FUNCTION_BLOCK fb_gm_operationElecylinder
VAR_INPUT
END_VAR
VAR_OUTPUT
END_VAR
VAR
	SFCInit: bool;
	TranPosDone: BOOL;
	TranNegDone: BOOL;
	flgInitDone: BOOL;
	PickUpPosDone: BOOL;
	PickUpNegDone: BOOL;
	var_process: INT;
END_VAR

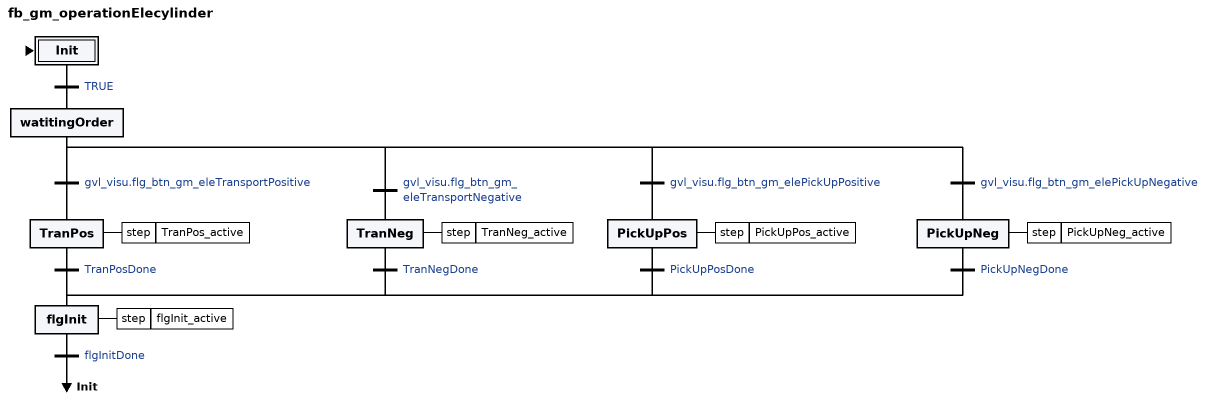
INITIAL_STEP Init:
END_STEP
TRANSITION FROM Init TO watitingOrder
    := TRUE;
END_TRANSITION
STEP watitingOrder:
END_STEP
TRANSITION FROM watitingOrder TO TranPos
    := gvl_visu.flg_btn_gm_eleTransportPositive;
END_TRANSITION
STEP TranPos:
    TranPos_active(N);  // step action
END_STEP
TRANSITION FROM TranPos TO flgInit
    := TranPosDone;
END_TRANSITION
TRANSITION FROM watitingOrder TO TranNeg
    := gvl_visu.flg_btn_gm_eleTransportNegative;
END_TRANSITION
STEP TranNeg:
    TranNeg_active(N);  // step action
END_STEP
TRANSITION FROM TranNeg TO flgInit
    := TranNegDone;
END_TRANSITION
TRANSITION FROM watitingOrder TO PickUpPos
    := gvl_visu.flg_btn_gm_elePickUpPositive;
END_TRANSITION
STEP PickUpPos:
    PickUpPos_active(N);  // step action
END_STEP
TRANSITION FROM PickUpPos TO flgInit
    := PickUpPosDone;
END_TRANSITION
TRANSITION FROM watitingOrder TO PickUpNeg
    := gvl_visu.flg_btn_gm_elePickUpNegative;
END_TRANSITION
STEP PickUpNeg:
    PickUpNeg_active(N);  // step action
END_STEP
TRANSITION FROM PickUpNeg TO flgInit
    := PickUpNegDone;
END_TRANSITION
STEP flgInit:
    flgInit_active(N);  // step action
END_STEP
TRANSITION FROM flgInit TO Init
    := flgInitDone;
END_TRANSITION

ACTION flgInit_active:
IF flgInit._x AND flgInit.x = FALSE THEN
	flgInitDone:= FALSE;
	gvl_visu.flg_btn_gm_eleTransportPositive := FALSE;
	gvl_visu.flg_btn_gm_eleTransportNegative := FALSE;
	gvl_visu.flg_btn_gm_elePickUpPositive := FALSE;
	gvl_visu.flg_btn_gm_elePickUpNegative := FALSE;
	gvl_visu.flg_btn_eleSamplePositive := FALSE;
	gvl_visu.flg_btn_eleSampleNegative := FALSE;
	gvl_visu.flg_btn_eleTrayChangePositive := FALSE;
	gvl_visu.flg_btn_eleTrayChangeNegative := FALSE;
	gvl_visu.flg_btn_eleRotaryPositive := FALSE;
	gvl_visu.flg_btn_eleRotaryNegative := FALSE;
ELSIF flgInit._x AND flgInit.x THEN
	flgInitDone := TRUE;
END_IF
END_ACTION

PROPERTY p_Init : bool
GET
p_init := THIS^.SFCInit;
END_GET
SET
THIS^.SFCInit := p_init;
END_SET
END_PROPERTY

ACTION PickUpNeg_active:
IF PickUpNeg._x AND PickUpNeg.x = FALSE THEN
	PickUpNegDone := FALSE;
	gvl_elecylinder.fbi_gm_axisPickUp.in_flg_run := FALSE;
	gvl_elecylinder.fbi_gm_axisPickUp.in_var_moveMode := eP_eleMoveMode.eleA;
	var_process := 0;
ELSIF PickUpNeg._x AND PickUpNeg.x THEN
	CASE var_process OF
		0:
			gvl_elecylinder.fbi_gm_axisPickUp.in_flg_run := TRUE;
			var_process := 1;
		1:
			IF gvl_elecylinder.fbi_gm_axisPickUp.out_flg_Done THEN
				gvl_elecylinder.fbi_gm_axisPickUp.in_flg_run := FALSE;
				PickUpNegDone := TRUE;
			END_IF
	END_CASE
END_IF
END_ACTION

ACTION PickUpPos_active:
IF PickUpPos._x AND PickUpPos.x = FALSE THEN
	PickUpPosDone := FALSE;
	gvl_elecylinder.fbi_gm_axisPickUp.in_flg_run := FALSE;
	gvl_elecylinder.fbi_gm_axisPickUp.in_var_moveMode := eP_eleMoveMode.eleB;
	var_process := 0;
ELSIF PickUpPos._x AND PickUpPos.x THEN
	CASE var_process OF
		0:
			gvl_elecylinder.fbi_gm_axisPickUp.in_flg_run := TRUE;
			var_process := 1;
		1:
			IF gvl_elecylinder.fbi_gm_axisPickUp.out_flg_Done THEN
				gvl_elecylinder.fbi_gm_axisPickUp.in_flg_run := FALSE;
				PickUpPosDone := TRUE;
			END_IF
	END_CASE
END_IF
END_ACTION

ACTION TranNeg_active:
IF TranNeg._x AND TranNeg.x = FALSE THEN
	TranNegDone := FALSE;
	gvl_elecylinder.fbi_gm_axisTransport.in_flg_run := FALSE;
	gvl_elecylinder.fbi_gm_axisTransport.in_var_moveMode := eP_eleMoveMode.eleA;
	var_process := 0;
ELSIF TranNeg._x AND TranNeg.x THEN
	CASE var_process OF
		0:
			gvl_elecylinder.fbi_gm_axisTransport.in_flg_run := TRUE;
			var_process := 1;
		1:
			IF gvl_elecylinder.fbi_gm_axisTransport.out_flg_Done THEN
				gvl_elecylinder.fbi_gm_axisTransport.in_flg_run := FALSE;
				TranNegDone := TRUE;
			END_IF
	END_CASE
END_IF
END_ACTION

ACTION TranPos_active:
IF TranPos._x AND TranPos.x = FALSE THEN
	TranPosDone := FALSE;
	gvl_elecylinder.fbi_gm_axisTransport.in_flg_run := FALSE;
	gvl_elecylinder.fbi_gm_axisTransport.in_var_moveMode := eP_eleMoveMode.eleB;
	var_process := 0;
ELSIF TranPos._x AND TranPos.x THEN
	CASE var_process OF
		0:
			gvl_elecylinder.fbi_gm_axisTransport.in_flg_run := TRUE;
			var_process := 1;
		1:
			IF gvl_elecylinder.fbi_gm_axisTransport.out_flg_Done THEN
				gvl_elecylinder.fbi_gm_axisTransport.in_flg_run := FALSE;
				TranPosDone := TRUE;
			END_IF
	END_CASE
END_IF
END_ACTION

END_FUNCTION_BLOCK

(* stored: Version 1.1.0.1, ProductVersion 3.1.4024.11
   POU fb_gm_operationElecylinder: Id {81da7721-46e3-4919-9f5c-c7ea16f238d2}, SpecialFunc None
   Action flgInit_active: Id {a160a8b8-43ef-4a74-800d-d552e8bef65b}
   Property p_Init: Id {36606747-d007-45db-bffc-48bc6670925e}
   Get Get: Id {318339dc-b7b1-47a1-8dea-73b6803dce21}
   Set Set: Id {61c8c1a4-f061-4939-8e50-71eaeb4eb30d}
   Action PickUpNeg_active: Id {77978a97-9522-472c-b6ec-366f96947542}
   Action PickUpPos_active: Id {73e98bcd-5321-4129-94a2-5f5b1b7a4700}
   Action TranNeg_active: Id {85a6cd7c-885a-4e73-8795-7874791a9f6f}
   Action TranPos_active: Id {721830da-6e18-4d9e-b048-9c80383c0f04} *)
